{attribute 'OPC.UA.DA.JobMethod' := 'JobMethode_CompressorControl'}
FUNCTION_BLOCK MBS_VSG_AS_VerticalMove
VAR
	AlwaysTrue : BOOL := TRUE;
	// Used for debugging purposes to display InputArguments of method call
	MethodCall_CompressorControl : BOOL := FALSE; // used to store InputArg "MethodCall" from Start() method
	Destination : BOOL;
	TS_EndschalterEntlastung : BOOL;
	callCounterStart : ULINT; // counts how many times the Start() method has been called
	callCounterCheckState : ULINT; // counts how many times the CheckState() method has been called
	callCounterAbort : ULINT; // counts how many times the Abort() method has been called
	
	// Variables to determine if a job has been started (Start() method has been called) or finished
	jobRunning : BOOL;
	jobFinished : BOOL;

	// State machine variable
	state : UDINT;
	
	//Variablen des Transport FBs
	ResetCall : BOOL := FALSE;	
	MBS_VSG_VerticalMove : CompressorControl;
END_VAR
	
VAR_INPUT
	NotAusSignal: BOOL;
//	LightSensor_01 : BOOL;
//	LightSensor_02 : BOOL;
	TS_Endschalter_01 : BOOL;
	TS_Endschalter_02 : BOOL;
	PowerOnDelay_Compressor : TIME;
	PowerOnDelay_Ventil : TIME;
END_VAR

VAR_OUTPUT
	Compressor : BOOL;
	Ventil : BOOL;
END_VAR

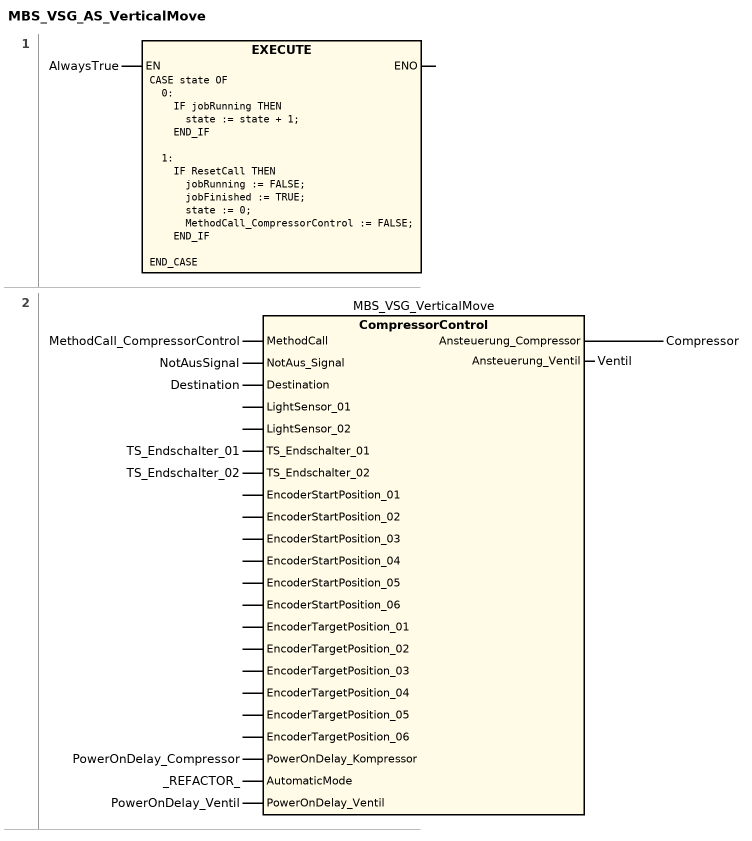
// NETWORK 1
IF AlwaysTrue THEN
    CASE state OF
    	0:
    		IF jobRunning THEN
    			state := state + 1;
    		END_IF
    		
    	1:
    		IF ResetCall THEN
    			jobRunning := FALSE;
    			jobFinished := TRUE;
    			state := 0;
    			MethodCall_CompressorControl := FALSE;
    		END_IF
    		
    END_CASE
END_IF

// NETWORK 2
MBS_VSG_VerticalMove(
    MethodCall := MethodCall_CompressorControl,
    NotAus_Signal := NotAusSignal,
    Destination := Destination,
    TS_Endschalter_01 := TS_Endschalter_01,
    TS_Endschalter_02 := TS_Endschalter_02,
    PowerOnDelay_Kompressor := PowerOnDelay_Compressor,
    AutomaticMode := _REFACTOR_,
    PowerOnDelay_Ventil := PowerOnDelay_Ventil,
    Ansteuerung_Ventil => Ventil); // CompressorControl
Compressor := MBS_VSG_VerticalMove.Ansteuerung_Compressor;

{attribute 'TcRpcEnable' := '1'}
METHOD Abort : HRESULT
VAR_INPUT
	hdl : UDINT; // Do not change, used by server.
END_VAR
callCounterAbort := callCounterAbort + 1;
END_METHOD

{attribute 'TcRpcEnable' := '1'}
METHOD CheckState : HRESULT
VAR_INPUT
	hdl : UDINT; // Do not change, used by server.
END_VAR
VAR_OUTPUT
	bBusy : BOOL; // Do not change. Used by server to find out if the job is finished
	
	// List of OutputArguments for OPC UA method, may be customized
	State : BOOL; // Abgeschlossener MethodCall
	MethodCall: BOOL; //Input Recall
END_VAR
callCounterCheckState := callCounterCheckState + 1;
IF NOT jobFinished THEN
	bBusy := TRUE; // job is not finished yet
	CheckState := 0; // no error
ELSE
	bBusy := FALSE; // job is finished
	CheckState := 0; // done, no error occured during execution (OPC UA StatusCode "GOOD")
	jobFinished := FALSE;
	State := ResetCall;
	MethodCall := MethodCall_CompressorControl;
END_IF
END_METHOD

{attribute 'TcRpcEnable' := '1'}
METHOD Start : HRESULT
VAR_INPUT
	// List of InputArguments for OPC UA method, may be customized
	MethodCall : BOOL; // some description
	Destination : BOOL;	
END_VAR
VAR_OUTPUT
	hdl : UDINT; // Do not change, used by server.
END_VAR
callCounterStart := callCounterStart + 1;

MethodCall_CompressorControl := MethodCall;
Destination := Destination;

jobRunning := TRUE;
Start := 0; // no error occured, e.g. while parsing the input arguments (0 = OPC UA StatusCode "GOOD")
END_METHOD

END_FUNCTION_BLOCK

(* stored: Version 1.1.0.1, ProductVersion 3.1.4024.15
   POU MBS_VSG_AS_VerticalMove: Id {95439bd0-2f49-4df3-96c4-b396d4584a44}, SpecialFunc None
   Method Abort: Id {2c3f2ec6-335d-4181-9ee3-b1ad2820bab5}
   Method CheckState: Id {cf469c2e-fa83-4ae0-9d55-c5b5ec7e6072}
   Method Start: Id {4a0cf284-944d-4a10-8697-8cdc626baa20} *)
